{attribute 'qualified_only'}
VAR_GLOBAL
	//master status
	//master status:type?

	//consider multi-master system from S7-300/400 systems
	
	//all slaves
	DPslaveDiag: ARRAY[1..maxNumDPSlaves] OF typeDPSlaveIndicator;

	//assign to mapped IO for DPstate
	RawDPStateDiag AT %I*: ARRAY[1..maxNumDPSlaves] OF USINT ;

END_VAR


VAR_GLOBAL CONSTANT
	maxNumDPSlaves: UINT := 127;
END_VAR


//refer to C79000-G8976-C124-03 04/2009

(* stored: Version 1.1.0.1, ProductVersion 3.1.4024.12
   GVL profibusDiag: Id {934ceea2-b1dd-4333-8f9b-25a929c1d377} *)
